# EPICS autosave request: softGlueApp/Db/softGlue_convenience_settings.req
$(P)$(H)busy.OUT
$(P)$(H)busy.FLNK
$(P)$(H)pulseOut.OUT
$(P)$(H)npulseOut.OUT
